(* IEC 61131-3 sources: plcassist-cli/packages/volt-lsp-iec/test-corpus/pro2193/Device/Plc Logic/Application/03 Hardware Units/31 SER/31.02 - X Units/Xu Unit for Chain, 3 files *)

(* ---- IXuUnit_ForChain_Config.itf ---- *)
// Commands specific for an Xu Unit
INTERFACE IXuUnit_ForChain_Config
EXTENDS IXuUnit_Default_Config

END_INTERFACE

(* ---- IXuUnit_ForChain_Transfer_Commands.itf ---- *)
// Commands specific for an Xu Unit
INTERFACE IXuUnit_ForChain_Transfer_Commands
EXTENDS IXuUnit_Default_Transfer_Commands, IModuleHasSafePosForChain

// Move to a position just before the chain
METHOD MoveToInFrontOfChain : BOOL
VAR_INPUT
END_VAR
END_METHOD

END_INTERFACE

(* ---- XuUnit_ForChainFB.fb ---- *)
{attribute 'symbol' := 'none'}
FUNCTION_BLOCK XuUnit_ForChainFB
EXTENDS XuUnit_DefaultFB
IMPLEMENTS IXuUnit_ForChain_Transfer_Commands, IXuUnit_ForChain_Config
VAR_IN_OUT
	DataProject					: XuUnit_ForChain_Data;
END_VAR
VAR
END_VAR
VAR CONSTANT
	rDistanceFromChain	: REAL := 25;
END_VAR

SUPER^(
	Data				:= Data,
	AxisRef				:= AxisRef,
	DataBrink			:= DataBrink,
	coveredDistance		:= coveredDistance,
);

END_FUNCTION_BLOCK

// Move to a position just before the chain
METHOD MoveToInFrontOfChain : BOOL
VAR_INPUT
END_VAR
%FOLDER Commands
IF NOT EnableHalfwayPosition THEN
	RETURN;
END_IF

IF HasPayload = enumPayload.None AND SER.OperationMode <> SER_OperationModeType.SemiAuto THEN
	RETURN;
END_IF

IF NOT CommandLock.Request(__POUNAME()) THEN
	RETURN;
END_IF

Drive.SetMovementProfileData(Data.Takeover[1]);

MoveToInFrontOfChain := Drive.MoveAbsPos(Data.Takeover[1].Pos.value - rDistanceFromChain);

CommandLock.Release(__POUNAME());
END_METHOD

// The X axis is homed, and in a safe (parking) position
{attribute 'monitoring':='call'}
PROPERTY PUBLIC InSafePosForChain : BOOL
%FOLDER Properties
GET
VAR
END_VAR
// Chain may already rotate when Xu unit is 15 mm back from Takeover pos
InSafePosForChain := movementInsideMouldActive OR_ELSE Drive.PosSmallerOrEqual(Data.Takeover[1].Pos.value - rDistanceFromChain) OR_ELSE InSafePos;

//InSafePosForChain := movementInsideMouldActive OR_ELSE Drive.PosSmallerOrEqual(Data.HalfwayPos.value) OR_ELSE InSafePos;
END_GET
END_PROPERTY
